// TIA Portal project "2022.05.28_第四章_移动指令" (V17)

(* hardware
DEVICE "S7-1500/ET200MP station_1"  S7-1500 station
   slot 0: "导轨_0"  Rack  6ES7 590-1***0-0AA0
   slot 1: "PLC_1500"  CPU 1516-3 PN/DP  6ES7 516-3AN00-0AB0  V1.7
      slot 3: "CPU 显示_1"  6ES7591-1BA00-0AA0
      slot 32768: "PROFINET 接口_1"  X1
         slot 32769: "端口_1"  X1 P1
         slot 32770: "端口_2"  X1 P2
      slot 33024: "PROFINET 接口_2"  X2
         slot 33025: "端口_1"  X2 P1
      slot 33280: "DP 接口_1"  X3
DEVICE "HMI_1"  TP1200 Comfort
   slot 0: "HMI_1"  TP1200 Comfort  6AV2 124-0MC01-0AX0  17.0.0.0
   slot 1: "HMI_RT_1"  TP1200 Comfort  6AV2 124-0MC01-0AX0  17.0.0.0
   slot 5: "HMI_1.IE_CP_1"  PROFINET Interface  17.0.0.0
      slot 1: "PROFINET Interface_1"  PROFINET Interface
         slot 1: "Port_1"  Port
         slot 2: "Port_2"  Port
   slot 7: "HMI_1.MPI/DP_CP_1"  MPI/DP Interface  17.0.0.0
*)

// ===== PLC "PLC_1500"  CPU 1516-3 PN/DP =====

TYPE "用户数据类型_1"
   STRUCT
      "a" : Int;
      "b" : Int;
      c : Int;
   END_STRUCT;
END_TYPE

DATA_BLOCK "DATE_AND_TIME"   // DB1
{ S7_Optimized_Access := 'TRUE' }
VERSION : 0.1
   VAR
      "time" : Date_And_Time;
      time_ret : Int;
   END_VAR
BEGIN
END_DATA_BLOCK

DATA_BLOCK "移动操作DB"   // DB2
{ S7_Optimized_Access := 'TRUE' }
VERSION : 0.1
   VAR
      移动块 : Struct
         移动块按钮 : Bool;
         IN : Array[0..10] of Int;
         OUT : Array[0..10] of Int;
      END_STRUCT;
      RET_VAL : Int;
      "B" : Array[0..10] of Int;
      "A" : Array[0..10] of Int;
      B_1 : Array[0..10] of "用户数据类型_1";
      A_1 : Array[0..10] of "用户数据类型_1";
      存储区移动 : Struct
         存储区移动按钮 : Bool;
         "A" : Array[0..10] of "用户数据类型_1";
         "B" : Array[0..10] of "用户数据类型_1";
      END_STRUCT;
      初始化 : Byte;
      移动值 : Struct
         "A" : Int;
         "B" : Int;
         移动值按钮 : Bool;
      END_STRUCT;
   END_VAR
BEGIN
END_DATA_BLOCK

FUNCTION "移动操作" : Void   // FC1, LAD
{ S7_Optimized_Access := 'TRUE' }
VERSION : 0.1
   VAR_TEMP   // added for the SCL form of the ladder/FBD networks
      _w1 : Bool;
   END_VAR
BEGIN

REGION Network 1: 移动值
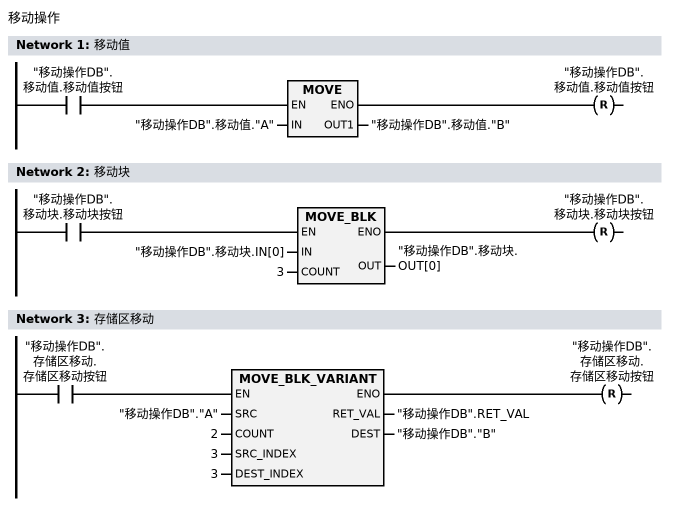
   RUNG wire#powerrail
      Contact( "移动操作DB".移动值.移动值按钮 )
      Move(in := "移动操作DB".移动值."A", out1 => "移动操作DB".移动值."B")
      R_Coil( "移动操作DB".移动值.移动值按钮 )
   END_RUNG
   // the same network as SCL:
   IF "移动操作DB".移动值.移动值按钮 THEN
       "移动操作DB".移动值."B" := "移动操作DB".移动值."A";
       "移动操作DB".移动值.移动值按钮 := FALSE;
   END_IF;
END_REGION

REGION Network 2: 移动块
   #_w1 := "移动操作DB".移动块.移动块按钮;
   IF #_w1 THEN
       MOVE_BLK(IN := "移动操作DB".移动块.IN[0], COUNT := 3, OUT => "移动操作DB".移动块.OUT[0]);
       "移动操作DB".移动块.移动块按钮 := FALSE;
   END_IF;
END_REGION

REGION Network 3: 存储区移动
   // ENO of a box is taken as its EN; it also drops when the box reports an error
   #_w1 := "移动操作DB".存储区移动.存储区移动按钮;
   IF #_w1 THEN
       "移动操作DB".RET_VAL := MOVE_BLK_VARIANT(SRC := "移动操作DB"."A",
                               COUNT := 2,
                               SRC_INDEX := 3,
                               DEST_INDEX := 3,
                               DEST => "移动操作DB"."B");
       "移动操作DB".存储区移动.存储区移动按钮 := FALSE;
   END_IF;
END_REGION
END_FUNCTION

FUNCTION "块_1" : Void   // FC2, SCL
{ S7_Optimized_Access := 'TRUE' }
VERSION : 0.1
BEGIN
   //移动值
   IF "移动操作DB".移动值.移动值按钮 THEN
       "移动操作DB".移动值.B := "移动操作DB".移动值.A;
       "移动操作DB".移动值.移动值按钮 := FALSE;
   END_IF;

   //移动块
   IF "移动操作DB".移动块.移动块按钮 THEN
       MOVE_BLK(IN:="移动操作DB".移动块.IN[0],
                COUNT:=3,
                OUT=>"移动操作DB".移动块.OUT[0]);
       "移动操作DB".移动块.移动块按钮 := FALSE;

   END_IF;

   //存储区移动
   IF "移动操作DB".存储区移动.存储区移动按钮 THEN
       "移动操作DB".存储区移动.RET_VAL := MOVE_BLK_VARIANT(SRC := "移动操作DB".A,
                                                  COUNT := 2,
                                                  SRC_INDEX := 3,
                                                  DEST_INDEX := 5,
                                                  DEST => "移动操作DB".B);
       "移动操作DB".存储区移动.存储区移动按钮 := FALSE;
   END_IF;
END_FUNCTION

ORGANIZATION_BLOCK "Main"   // OB1, LAD, ProgramCycle
TITLE = "Main Program Sweep (Cycle)"
{ S7_Optimized_Access := 'TRUE' }
VERSION : 0.1
   VAR_INPUT
      Initial_Call : Bool;   // Initial call of this OB
      Remanence : Bool;   // =True, if remanent data are available
   END_VAR
BEGIN

REGION Network 1
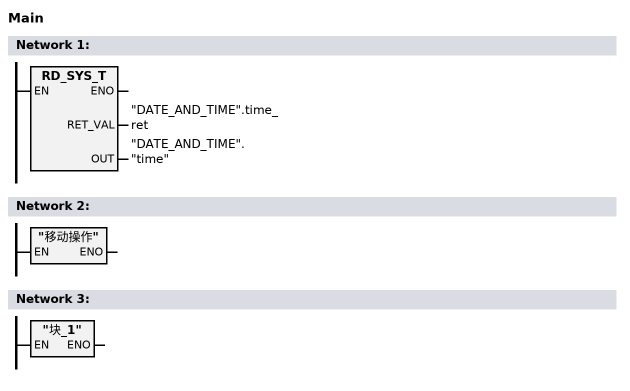
   "DATE_AND_TIME".time_ret := RD_SYS_T(OUT => "DATE_AND_TIME"."time");
END_REGION

REGION Network 2
   RUNG wire#powerrail
      "移动操作"()
   END_RUNG
   // the same network as SCL:
   "移动操作"();
END_REGION

REGION Network 3
   RUNG wire#powerrail
      "块_1"()
   END_RUNG
   // the same network as SCL:
   "块_1"();
END_REGION
END_ORGANIZATION_BLOCK

(* ===== HMI "HMI_RT_1" =====
system functions are stored by id; their names below are inferred from use
connection "PLC_1500": ETHERNET, S7_1500_OMS
connection "Connection_1": ETHERNET, S7_1500_OMS

HMI tags "默认变量表"
   "DATE_AND_TIME_time_ret" : Int = PLC "DATE_AND_TIME".time_ret, 1 s
   "移动操作DB_移动值_移动值按钮" : Bool = PLC 移动操作DB.移动值.移动值按钮, 1 s
   "移动操作DB_移动值_A" : Int = PLC 移动操作DB.移动值.A, 1 s
   "移动操作DB_移动值_B" : Int = PLC 移动操作DB.移动值.B, 1 s
   "移动操作DB_移动块_IN{0}" : Int = PLC 移动操作DB.移动块.IN[0], 1 s
   "移动操作DB_移动块_IN{1}" : Int = PLC 移动操作DB.移动块.IN[1], 1 s
   "移动操作DB_移动块_IN{2}" : Int = PLC 移动操作DB.移动块.IN[2], 1 s
   "移动操作DB_移动块_OUT{0}" : Int = PLC 移动操作DB.移动块.OUT[0], 1 s
   "移动操作DB_移动块_OUT{1}" : Int = PLC 移动操作DB.移动块.OUT[1], 1 s
   "移动操作DB_移动块_OUT{2}" : Int = PLC 移动操作DB.移动块.OUT[2], 1 s
   "移动操作DB_移动块_移动块按钮" : Bool = PLC 移动操作DB.移动块.移动块按钮, 1 s
   "移动操作DB_A{0}" : Int = PLC 移动操作DB.A[0], 1 s
   "移动操作DB_A{1}" : Int = PLC 移动操作DB.A[1], 1 s
   "移动操作DB_A_1{0}_a" : Int = PLC 移动操作DB.A_1[0].a, 1 s
   "移动操作DB_A_1{0}_b" : Int = PLC 移动操作DB.A_1[0].b, 1 s
   "移动操作DB_A_1{0}_c" : Int = PLC 移动操作DB.A_1[0].c, 1 s
   "移动操作DB_A_1{1}_a" : Int = PLC 移动操作DB.A_1[1].a, 1 s
   "移动操作DB_A_1{1}_b" : Int = PLC 移动操作DB.A_1[1].b, 1 s
   "移动操作DB_A_1{1}_c" : Int = PLC 移动操作DB.A_1[1].c, 1 s
   "移动操作DB_B_1{1}_a" : Int = PLC 移动操作DB.B_1[1].a, 1 s
   "移动操作DB_B_1{1}_b" : Int = PLC 移动操作DB.B_1[1].b, 1 s
   "移动操作DB_B_1{1}_c" : Int = PLC 移动操作DB.B_1[1].c, 1 s
   "移动操作DB_B_1{2}_a" : Int = PLC 移动操作DB.B_1[2].a, 1 s
   "移动操作DB_B_1{2}_b" : Int = PLC 移动操作DB.B_1[2].b, 1 s
   "移动操作DB_B_1{2}_c" : Int = PLC 移动操作DB.B_1[2].c, 1 s
   "移动操作DB_存储区移动按钮" :  = PLC 移动操作DB.存储区移动, 1 s

HMI tags "外部变量"
   "DATE_AND_TIME_time" : Date_And_Time = PLC "DATE_AND_TIME".time, 1 s

HMI tags "内部变量"
   "画面切换颜色" : Int, internal

screen "首页" 1280x740, template "模板_1"
   on GenerateScreen: SetTag("画面切换颜色", 1)

Template "模板_1" 1280x740
   Button "Template_Button_13" at 81,679 size 153x59; TextOff '用户界面1'
      on Release: ActivateScreen("用户界面1", 0); SetTag("画面切换颜色", 2)
      Appearance <- "画面切换颜色"
   Button "退出" at 1200,679 size 78x59; TextOff '退出'; PictureOff "ExitRuntime_TP1200_Comfort_TR"; PictureOn "ExitRuntime_TP1200_Comfort_TR"
      on Release: StopRuntime(0)
   Button "起始画面" at 1,679 size 78x59; TextOff '起始画面'; PictureOff "NavigateHome_TP1200_Comfort_TR"; PictureOn "NavigateHome_TP1200_Comfort_TR"
      on Release: SetTag("画面切换颜色", 1); ActivateScreen("首页", 0)
      Appearance <- "画面切换颜色"
   Button "Template_Button_1" at 236,679 size 153x59; TextOn '用户界面2'; TextOff '用户界面2'
      on Release: ActivateScreen("用户界面2", 0); SetTag("画面切换颜色", 3)
      Appearance <- "画面切换颜色"
   Button "Template_Button_2" at 393,678 size 153x59; TextOn '测试界面'; TextOff '测试界面'
      on Release: ActivateScreen("测试界面", 0); SetTag("画面切换颜色", 4)
      Appearance <- "画面切换颜色"
   Button "Template_Button_3" at 551,678 size 153x59; TextOn '用户管理界面'; TextOff '用户管理界面'
      on Release: ActivateScreen("用户管理界面", 0); SetTag("画面切换颜色", 5)
      Appearance <- "画面切换颜色"
   Button "Template_Button_4" at 710,678 size 153x59; TextOn '报警管理界面'; TextOff '报警管理界面'
      on Release: ActivateScreen("报警视图画面", 0); SetTag("画面切换颜色", 6)
      Appearance <- "画面切换颜色"
   Button "Template_Button_5" at 868,678 size 153x59; TextOn '系统诊断界面'; TextOff '系统诊断界面'
      on Release: ActivateScreen("系统诊断界面", 0); SetTag("画面切换颜色", 7)
      Appearance <- "画面切换颜色"
   Button "Template_Button_6" at 1027,678 size 153x59; TextOn '备用界面'; TextOff '备用界面'
      on Release: ActivateScreen("备用界面", 0); SetTag("画面切换颜色", 8)
      Appearance <- "画面切换颜色"

screen "用户界面1" 1280x740, template "模板_1"
   Button "按钮_1" at 281,126 size 96x43; TextOff '移动'
      on Press: SetBit("移动操作DB_移动值_移动值按钮")
   IOField "I/O 域_1" at 417,130 size 96x43; FormatPattern s99999
      ProcessValue <- "移动操作DB_移动值_B"
   IOField "I/O 域_2" at 145,126 size 96x43; FormatPattern s99999
      ProcessValue <- "移动操作DB_移动值_A"
   TextField "文本域_1" at 276,98 size 95x21; Text '移动值指令'
   Button "按钮_2" at 281,364 size 96x43; TextOff '移动'
      on Press: SetBit("移动操作DB_移动块_移动块按钮")
   IOField "I/O 域_3" at 417,293 size 96x43; FormatPattern s99999
      ProcessValue <- "移动操作DB_移动块_OUT{0}"
   IOField "I/O 域_4" at 145,289 size 96x43; FormatPattern s99999
      ProcessValue <- "移动操作DB_移动块_IN{0}"
   TextField "文本域_2" at 276,261 size 95x21; Text '移动块指令'
   IOField "I/O 域_5" at 417,363 size 96x43; FormatPattern s99999
      ProcessValue <- "移动操作DB_移动块_OUT{1}"
   IOField "I/O 域_6" at 145,359 size 96x43; FormatPattern s99999
      ProcessValue <- "移动操作DB_移动块_IN{1}"
   IOField "I/O 域_7" at 417,433 size 96x43; FormatPattern s99999
      ProcessValue <- "移动操作DB_移动块_OUT{2}"
   IOField "I/O 域_8" at 145,429 size 96x43; FormatPattern s99999
      ProcessValue <- "移动操作DB_移动块_IN{2}"
   Button "按钮_3" at 701,416 size 96x43; TextOff '移动'
      on Press: SetBit("移动操作DB_存储区移动按钮")
   TextField "文本域_3" at 696,261 size 131x21; Text '存储区移动按钮'
   IOField "I/O 域_9" at 571,293 size 96x32; FormatPattern s99999
      ProcessValue <- "移动操作DB_A_1{0}_a"
   IOField "I/O 域_10" at 571,345 size 96x32; FormatPattern s99999
      ProcessValue <- "移动操作DB_A_1{0}_b"
   IOField "I/O 域_11" at 571,397 size 96x32; FormatPattern s99999
      ProcessValue <- "移动操作DB_A_1{0}_c"
   IOField "I/O 域_12" at 571,449 size 96x32; FormatPattern s99999
      ProcessValue <- "移动操作DB_A_1{1}_a"
   IOField "I/O 域_13" at 571,501 size 96x32; FormatPattern s99999
      ProcessValue <- "移动操作DB_A_1{1}_b"
   IOField "I/O 域_14" at 571,554 size 96x32; FormatPattern s99999
      ProcessValue <- "移动操作DB_A_1{1}_c"
   IOField "I/O 域_15" at 837,293 size 96x32; FormatPattern s99999
      ProcessValue <- "移动操作DB_B_1{1}_a"
   IOField "I/O 域_16" at 837,345 size 96x32; FormatPattern s99999
      ProcessValue <- "移动操作DB_B_1{1}_b"
   IOField "I/O 域_17" at 837,397 size 96x32; FormatPattern s99999
      ProcessValue <- "移动操作DB_B_1{1}_c"
   IOField "I/O 域_18" at 837,449 size 96x32; FormatPattern s99999
      ProcessValue <- "移动操作DB_B_1{2}_a"
   IOField "I/O 域_19" at 837,501 size 96x32; FormatPattern s99999
      ProcessValue <- "移动操作DB_B_1{2}_b"
   IOField "I/O 域_20" at 837,554 size 96x32; FormatPattern s99999
      ProcessValue <- "移动操作DB_B_1{2}_c"

screen "用户管理界面" 1280x740, template "模板_1"
   UserView "用户视图_1" at 2,2 size 1277x676

screen "报警视图画面" 1280x740, template "模板_1"
   AlarmView "报警视图_1" at 0,0 size 1280x676

screen "系统诊断界面" 1280x740, template "模板_1"
   SysDiagControl "系统诊断视图_1" at 0,2 size 1278x676
*)